{attribute addProperty BoxType "AX8620-0000-0026"}
{attribute addProperty Id "StatuswordAT %I*Statusword_3B58AC51162"}
{attribute addProperty CRC "854043290"}
{attribute addProperty SizeInBites "16"}
{attribute addProperty SizeInBytes "2"}
TYPE PSM_Statusword_32E7AA9A :
STRUCT
	{attribute addProperty Name "Statusword"}
	Statusword AT %I* : Statusword_3B58AC51;
END_STRUCT
END_TYPE

(* stored: Version 1.2.0.0, ProductVersion 3.1.4024.9
   DUT PSM_Statusword_32E7AA9A: Id {23bbf2c8-47e9-45b2-a85b-4c3d8cb050b8} *)
